// TIA Portal V18 export
FUNCTION_BLOCK "shutter"   // FB42, FBD
{ S7_Optimized_Access := 'TRUE' }
VERSION : 0.1
// stored: AutoNumber true, IsIECCheckEnabled false, IsRetainMemResEnabled false, MemoryReserve 100, SetENOAutomatically false, UDAEnableTagReadback false
   VAR_INPUT
      "allowed OPEN" : Bool := true;
      xbh_close : Bool;
      xSensClosed : Bool;
      xSensOpen : Bool;
      pt_val : Time := T#3s;
   END_VAR
   VAR_OUTPUT
      yPneumClose : Bool;
      er_no_closing : Bool;
      er_no_opening : Bool;
      er_both_activated : Bool;
   END_VAR
   VAR
      tonclos { S7_SetPoint := 'True'} : TON_TIME;
      tonopn { S7_SetPoint := 'True'} : TON_TIME;
   END_VAR
   VAR RETAIN
      commandClose : Bool;
   END_VAR
   VAR
      mem : Bool;
   END_VAR
   VAR_TEMP
      btn_clk : Bool;
   END_VAR
BEGIN

REGION Network 1
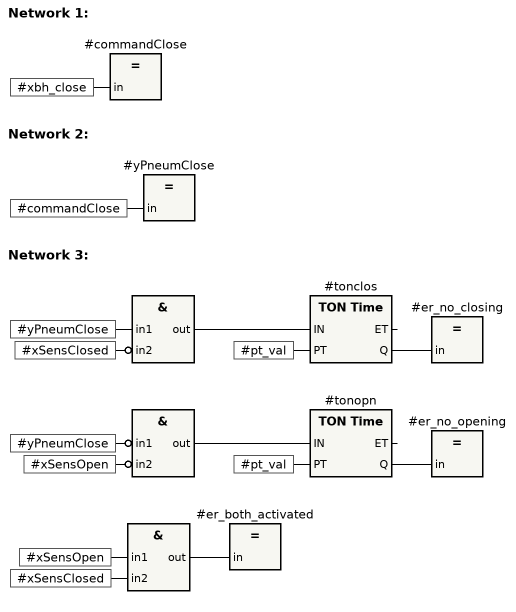
   #commandClose := #xbh_close;
END_REGION

REGION Network 2
   #yPneumClose := #commandClose;
END_REGION

REGION Network 3
   #tonclos(IN := #yPneumClose AND NOT #xSensClosed, PT := #pt_val);   // TON
   #er_no_closing := #tonclos.Q;
   #tonopn(IN := NOT #yPneumClose AND NOT #xSensOpen, PT := #pt_val);   // TON
   #er_no_opening := #tonopn.Q;
   #er_both_activated := #xSensOpen AND #xSensClosed;
END_REGION
END_FUNCTION_BLOCK
